// TIA Portal V20 export
TYPE "LER_typeServoPressTrackingData"
// stored: Access Published
   STRUCT
      "pvCurveYMAX-X" { ExternalWritable := 'False'} : Real;
      "pvCurveYMAX-Y" { ExternalWritable := 'False'} : Real;
      resultOK { ExternalWritable := 'False'} : Bool;
      resultNG { ExternalWritable := 'False'} : Bool;
      complete { ExternalWritable := 'False'} : Bool;
   END_STRUCT;
END_TYPE
